  [1568] = {x=211, y=-48.066, z=198, rx=180, rz=-90, shoulder=lefty, elbow=epositive, wrist=wpositive, fatherId=fReference[0]}
  [1569] = {x=211, y=-58.12, z=198, rx=180, rz=-90, shoulder=lefty, elbow=epositive, wrist=wpositive, fatherId=fReference[0]}
  [1570] = {x=211, y=-68.173, z=198, rx=180, rz=-90, shoulder=lefty, elbow=epositive, wrist=wpositive, fatherId=fReference[0]}
  [1571] = {x=211, y=-78.226, z=198, rx=180, rz=-90, shoulder=lefty, elbow=epositive, wrist=wpositive, fatherId=fReference[0]}
  [1572] = {x=211, y=-88.28, z=198, rx=180, rz=-90, shoulder=lefty, elbow=epositive, wrist=wpositive, fatherId=fReference[0]}
  [1573] = {x=211, y=-98.333, z=198, rx=180, rz=-90, shoulder=lefty, elbow=epositive, wrist=wpositive, fatherId=fReference[0]}
  [1574] = {x=211, y=-108.386, z=198, rx=180, rz=-90, shoulder=lefty, elbow=epositive, wrist=wpositive, fatherId=fReference[0]}
  [1575] = {x=211, y=-118.44, z=198, rx=180, rz=-90, shoulder=lefty, elbow=epositive, wrist=wpositive, fatherId=fReference[0]}
  [1576] = {x=211, y=-128.493, z=198, rx=180, rz=-90, shoulder=lefty, elbow=epositive, wrist=wpositive, fatherId=fReference[0]}
  [1577] = {x=211, y=-138.546, z=198, rx=180, rz=-90, shoulder=lefty, elbow=epositive, wrist=wpositive, fatherId=fReference[0]}
  [1578] = {x=211, y=-148.6, z=198, rx=180, rz=-88.43, shoulder=lefty, elbow=epositive, wrist=wpositive, fatherId=fReference[0]}
  [1579] = {x=210.725, y=-158.644, z=198, rx=180, rz=-79.45, shoulder=lefty, elbow=epositive, wrist=wpositive, fatherId=fReference[0]}
  [1580] = {x=208.886, y=-168.515, z=198, rx=180, rz=-69.519, shoulder=lefty, elbow=epositive, wrist=wpositive, fatherId=fReference[0]}
  [1581] = {x=205.373, y=-177.921, z=198, rx=180, rz=-59.588, shoulder=lefty, elbow=epositive, wrist=wpositive, fatherId=fReference[0]}
  [1582] = {x=200.29, y=-186.58, z=198, rx=180, rz=-49.656, shoulder=lefty, elbow=epositive, wrist=wpositive, fatherId=fReference[0]}
  [1583] = {x=193.79, y=-194.233, z=198, rx=-180, rz=-39.725, shoulder=lefty, elbow=epositive, wrist=wpositive, fatherId=fReference[0]}
  [1584] = {x=186.068, y=-200.65, z=198, rx=180, rz=-29.794, shoulder=lefty, elbow=epositive, wrist=wpositive, fatherId=fReference[0]}
  [1585] = {x=177.354, y=-205.639, z=198, rx=-180, rz=-19.863, shoulder=lefty, elbow=epositive, wrist=wpositive, fatherId=fReference[0]}
  [1586] = {x=167.911, y=-209.051, z=198, rx=180, rz=-9.931, shoulder=lefty, elbow=epositive, wrist=wpositive, fatherId=fReference[0]}
  [1587] = {x=158.02, y=-210.782, z=198, rx=-180, rz=-1.241, shoulder=lefty, elbow=epositive, wrist=wpositive, fatherId=fReference[0]}
  [1588] = {x=147.973, y=-211, z=198, rx=-180, shoulder=lefty, elbow=epositive, wrist=wpositive, fatherId=fReference[0]}
  [1589] = {x=137.92, y=-211, z=198, rx=180, shoulder=lefty, elbow=epositive, wrist=wpositive, fatherId=fReference[0]}
  [1590] = {x=127.867, y=-211, z=198, rx=180, shoulder=lefty, elbow=epositive, wrist=wpositive, fatherId=fReference[0]}
  [1591] = {x=117.813, y=-211, z=198, rx=-180, shoulder=lefty, elbow=epositive, wrist=wpositive, fatherId=fReference[0]}
  [1592] = {x=107.76, y=-211, z=198, rx=180, shoulder=lefty, elbow=epositive, wrist=wpositive, fatherId=fReference[0]}
  [1593] = {x=97.707, y=-211, z=198, rx=180, shoulder=lefty, elbow=epositive, wrist=wpositive, fatherId=fReference[0]}
  [1594] = {x=87.653, y=-211, z=198, rx=-180, shoulder=lefty, elbow=epositive, wrist=wpositive, fatherId=fReference[0]}
  [1595] = {x=77.6, y=-211, z=198, rx=-180, shoulder=lefty, elbow=epositive, wrist=wpositive, fatherId=fReference[0]}
  [1596] = {x=67.547, y=-211, z=198, rx=-180, shoulder=lefty, elbow=epositive, wrist=wpositive, fatherId=fReference[0]}
  [1597] = {x=57.493, y=-211, z=198, rx=-180, shoulder=lefty, elbow=epositive, wrist=wpositive, fatherId=fReference[0]}
  [1598] = {x=47.44, y=-211, z=198, rx=180, shoulder=lefty, elbow=epositive, wrist=wpositive, fatherId=fReference[0]}
  [1599] = {x=37.387, y=-211, z=198, rx=-180, shoulder=lefty, elbow=epositive, wrist=wpositive, fatherId=fReference[0]}
  [1600] = {x=27.333, y=-211, z=198, rx=180, shoulder=lefty, elbow=epositive, wrist=wpositive, fatherId=fReference[0]}
  [1601] = {x=17.28, y=-211, z=198, rx=180, shoulder=lefty, elbow=epositive, wrist=wpositive, fatherId=fReference[0]}
  [1602] = {x=7.227, y=-211, z=198, rx=180, shoulder=lefty, elbow=epositive, wrist=wpositive, fatherId=fReference[0]}
  [1603] = {x=-2.826, y=-211, z=198, rx=-180, shoulder=lefty, elbow=epositive, wrist=wpositive, fatherId=fReference[0]}
  [1604] = {x=-12.88, y=-211, z=198, rx=180, shoulder=lefty, elbow=epositive, wrist=wpositive, fatherId=fReference[0]}
  [1605] = {x=-22.933, y=-211, z=198, rx=180, shoulder=lefty, elbow=epositive, wrist=wpositive, fatherId=fReference[0]}
  [1606] = {x=-32.986, y=-211, z=198, rx=-180, shoulder=lefty, elbow=epositive, wrist=wpositive, fatherId=fReference[0]}
  [1607] = {x=-43.04, y=-211, z=198, rx=-180, shoulder=lefty, elbow=epositive, wrist=wpositive, fatherId=fReference[0]}
  [1608] = {x=-53.093, y=-211, z=198, rx=-180, shoulder=lefty, elbow=epositive, wrist=wpositive, fatherId=fReference[0]}
  [1609] = {x=-63.146, y=-211, z=198, rx=-180, shoulder=lefty, elbow=epositive, wrist=wpositive, fatherId=fReference[0]}
  [1610] = {x=-73.2, y=-211, z=198, rx=-180, shoulder=lefty, elbow=epositive, wrist=wpositive, fatherId=fReference[0]}
  [1611] = {x=-83.253, y=-211, z=198, rx=180, shoulder=lefty, elbow=epositive, wrist=wpositive, fatherId=fReference[0]}
  [1612] = {x=-93.306, y=-211, z=198, rx=180, shoulder=lefty, elbow=epositive, wrist=wpositive, fatherId=fReference[0]}
  [1613] = {x=-103.36, y=-211, z=198, rx=-180, shoulder=lefty, elbow=epositive, wrist=wpositive, fatherId=fReference[0]}
  [1614] = {x=-113.413, y=-211, z=198, rx=-180, shoulder=lefty, elbow=epositive, wrist=wpositive, fatherId=fReference[0]}
  [1615] = {x=-123.466, y=-211, z=198, rx=180, shoulder=lefty, elbow=epositive, wrist=wpositive, fatherId=fReference[0]}
  [1616] = {x=-133.52, y=-211, z=198, rx=180, shoulder=lefty, elbow=epositive, wrist=wpositive, fatherId=fReference[0]}
  [1617] = {x=-143.573, y=-211, z=198, rx=180, rz=0.019, shoulder=lefty, elbow=epositive, wrist=wpositive, fatherId=fReference[0]}
  [1618] = {x=-153.626, y=-210.997, z=198, rx=-180, rz=5.584, shoulder=lefty, elbow=epositive, wrist=wpositive, fatherId=fReference[0]}
  [1619] = {x=-163.619, y=-210.02, z=198, rx=-180, rz=15.516, shoulder=lefty, elbow=epositive, wrist=wpositive, fatherId=fReference[0]}
  [1620] = {x=-173.294, y=-207.334, z=198, rx=-180, rz=25.447, shoulder=lefty, elbow=epositive, wrist=wpositive, fatherId=fReference[0]}
  [1621] = {x=-182.361, y=-203.019, z=198, rx=180, rz=35.378, shoulder=lefty, elbow=epositive, wrist=wpositive, fatherId=fReference[0]}
  [1622] = {x=-190.548, y=-197.206, z=198, rx=-180, rz=45.309, shoulder=lefty, elbow=epositive, wrist=wpositive, fatherId=fReference[0]}
  [1623] = {x=-197.609, y=-190.068, z=198, rx=180, rz=55.241, shoulder=lefty, elbow=epositive, wrist=wpositive, fatherId=fReference[0]}
  [1624] = {x=-203.334, y=-181.819, z=198, rx=-180, rz=65.172, shoulder=lefty, elbow=epositive, wrist=wpositive, fatherId=fReference[0]}
  [1625] = {x=-207.55, y=-172.706, z=198, rx=-180, rz=75.103, shoulder=lefty, elbow=epositive, wrist=wpositive, fatherId=fReference[0]}
  [1626] = {x=-210.131, y=-163.003, z=198, rx=-180, rz=85.034, shoulder=lefty, elbow=epositive, wrist=wpositive, fatherId=fReference[0]}
  [1627] = {x=-211, y=-153, z=198, rx=-180, rz=85.034, shoulder=lefty, elbow=epositive, wrist=wpositive, fatherId=fReference[0]}
  [1628] = {x=-211, y=-153, z=198, rx=-180, rz=85.034, shoulder=lefty, elbow=epositive, wrist=wpositive, fatherId=fReference[0]}
  [1629] = {x=-211, y=-153, z=298, rx=-180, rz=85.034, shoulder=lefty, elbow=epositive, wrist=wpositive, fatherId=fReference[0]}
public tool tTool = {z=452, fatherId=flange[0], ioLink=valve1}
aio Tpompe = {link=CanIO\RemIO\remio0_QW}
dio doValve1 = {link=valve1}
